PROGRAM PRG_CNCAxesHandler
VAR
	nHliAxisIdx					: INT;				
	fbCNC_Axis					: ARRAY[0..HLI_SYS_AX_MAXIDX] OF HLI3_CNCAxis;;	
	
	nFirstSpindle				: INT := -1;
	fbHandleSpindleTechno		: HLI3_HandleSpindleTechnoGearChange;
	M3,M4,M5,M19				: BOOL;
	MDummy						: BOOL;
	M40, M41, M42, M43, M44, M45: BOOL;
		
	// FB_CNCAxis Sample
	// fbAxis_X 					:  FB_CNCAxis; 
	// stParameter					:  ST_CNC_AX_Parameter;
	// stOptions					:  ST_CNC_AX_Options;
	// stPLCopen					:  ST_CNC_AX_PLCopen;
			
	(*
	fbHandleSpindleTechnoPlcSp	: HLI3_HandleSpindleTechno;
	SM3,SM4,SM5,SM19			: bool; 
	*)
	bCalibrationCam: BOOL;
END_VAR

(****************************************************************************************)
(* POU:		PRG_AxesHandler                     										*)
(* Type:	PRG																			*)
(* Author: 	TV,MiB                                             							*)
(* Date: 	15.02.2018																	*)
(* Rev.: 	1.4                                               							*)
(* ------------------------------------------------------------------------------------ *)
(* Desc:	Description																	*)
(****************************************************************************************)

(****************************************************************************************)
(*							Release of all reachable axes								*)
(****************************************************************************************)

FOR nHliAxisIdx := 0 TO UDINT_TO_INT(gNrAx-1) DO
		
	fbCNC_Axis[nHliAxisIdx](
		nHliAxisIdx := nHliAxisIdx,		
		bEnable		:= PLCAxisEnable);
	
		IF HLI3_CheckAxisValid(nHliAxisIdx) THEN
			IF nFirstSpindle = -1 AND gpAx[nHliAxisIdx]^.ipo_state.spindle_axis_r THEN  (* store HLIIndex of first spindle *)
				nFirstSpindle := nHliAxisIdx;
			END_IF
		END_IF
END_FOR


	// FB_CNCAxis Sample 

	// CNC Axis Options
	
	// stOptions.strPathCompTable;
	// stOptions.bActivateCompTable;
	// stOptions.bProbingSignal;
	// stOptions.bReducedSpeed;
	// stOptions.bReducedSpeedZone1;
	// stOptions.bReducedSpeedZone2;
	// stOptions.bResetCalibration;
	
	// CNC Parameters
			
	// stParameter.bWriteParameter;
	// stParameter.nNumParameters  	:= 2;
	// stParameter.strTempPath		:= 'C:\';
	
	// stParameter.ParamList[0].strName 	:= 'kenngr.swe_pos';
	// stParameter.ParamList[0].strValue 	:= '30000000';

	// stParameter.ParamList[1].strName 	:= 'kenngr.swe_neg';
	// stParameter.ParamList[1].strValue 	:= '0';

	// PLCOpen
	// stPLCopen.nOverride;
	// stPLCopen.bExecuteHoming;
	// stPLCopen.bCamSignal;
	// stPLCopen.bExecuteMoveAbsolute;
	// stPLCopen.bExecuteReset;
	// stPLCopen.fPosition;
	// stPLCopen.fVelocity;
	// stPLCopen.fAcceleration;
	// stPLCopen.fJerk;
	
	(*
	fbAxis_X(
		nLogAxisNo:=1, 
		bEnable:= PLCAxisEnable, 
		bCalibrationCam:= bCalibrationCam, 
		bSetRefOffset:= , 
		fRefOffset:= , 
		stOptions:= stOptions, 
		stParameter:= stParameter, 
		stPLCopen:= stPLCopen, 
		stStatus=> );
*)		
 

(* if there exits spindles use the first one for spindleoverride *)
IF nFirstSpindle <> -1 THEN
	HLI3_SetAxisOverride(nHliAxisIdx:= nFirstSpindle , nOverride:= PLCSpindleOverride *10);

	fbHandleSpindleTechno(
		nHliAxisIdx:=nFirstSpindle , 		
		bIsChannelSpecific:= FALSE, 
		nRevolution=> , 
		nPosition=> , 
		bError=> , 
		nErrorId=> , 
		M03:= M3, 
		M04:= M4, 
		M05:= M5, 
		M19:= M19,
		M40 := M40,
		M41 := M41,
		M42 := M42,
		M43 := M43,
		M44 := M44,
		M45 := M45,
		); 
	(* acknowledge all spindle M funnctions immediately *)
	M3 := FALSE;  
	M4 := FALSE;
	M5 := FALSE;
	M19 := FALSE;
END_IF



(* Howto use plc controlled spindle : *)
(*
fbHandleSpindleTechnoPlcSp(
	nHliAxisIdx:= 0 , 
	nHliChannelIdx:= 0 , 
	bIsChannelSpecific:= TRUE, 
	nLogAxisNoChannelSpecific:= 95 , 
	bHandleGearChange:= FALSE , 
	bChannelReset:= FALSE, 
	nRevolution=> , 
	nPosition=> , 
	bError=> , 
	nErrorId=> , 
	M03:= SM3, 
	M04:= SM4, 
	M05:= SM5, 
	M19:= SM19);
*)

END_PROGRAM

(* stored: Version 1.1.0.1, ProductVersion 3.1.4022.9
   POU PRG_CNCAxesHandler: Id {09e86179-f0c7-4e63-9c4c-17d3691b5ccb}, SpecialFunc None *)
